PROGRAM MAP_IN
VAR

  {attribute 'TcLinkTo' := '._by := TIPC^XtsTransport^XtsTransport Instance^PlcTask Outputs^MAP_OUT.uTransportState._by'}
  uTransportState     : U_XTS_TRANSPORT_STATE;
  {attribute 'TcLinkTo' := '._by := TIPC^XtsTransport^XtsTransport Instance^PlcTask Outputs^MAP_OUT.uStationState._by'}
  uStationState       : U_STATION_STATE;
END_VAR

          // destination address
                                            // source address
                                                                    // size
  memcpy(ADR(GVL_XTS.XtsTransportState),  ADR(uTransportState),   SIZEOF(ST_XTS_TRANSPORT_STATE));
  memcpy(ADR(GVL_XTS.StationState),       ADR(uStationState),     SIZEOF(uStationState));

END_PROGRAM

(* stored: Version 1.1.0.1, ProductVersion 3.1.4024.12
   POU MAP_IN: Id {fbb445d4-48c0-4c41-ac0e-76f242f6b4cd}, SpecialFunc None *)
